TYPE
    InputBase_8311D824 :
    STRUCT
    END_STRUCT
END_TYPE

(* stored: Version 1.1.0.1, ProductVersion 3.1.4024.12
   DUT InputBase_8311D824: Id {f11a92e3-1782-0ab2-2cec-a1d3406e6d77} *)
